{attribute 'GeneratedUsingTerminal: EK1122-0000-0018'}
{attribute addProperty BoxType "EK1122-0000-0018"}
{attribute addProperty Id "Beckhoff_EL6xxxsub_EK1100EK1100_AB5A94672"}
{attribute addProperty CRC "1483390984"}
{attribute addProperty Size "2"}
TYPE Beckhoff_EL6xxxEK1122_586AC008 EXTENDS EK1122_AB5A9467 :
STRUCT
	{attribute addProperty Name "Beckhoff_EL6xxxsub_EK1100"}
	Beckhoff_EL6xxxsub_EK1100 : EK1100_AB5A9467;
END_STRUCT
END_TYPE

(* stored: Version 1.2.0.0, ProductVersion 3.1.4024.9
   DUT Beckhoff_EL6xxxEK1122_586AC008: Id {0acc8b5d-8af1-4d8f-a5df-b1ada3a18071} *)
